// SIMATIC S7-200 SMART project (STEP 7-Micro/WIN SMART), CPU SR40

SYMBOL_TABLE 系统符号
Always_On        SM0.0    // 始终接通
Clock_1s         SM0.5    // 针对 1 s 的周期时间，时钟脉冲接通 0.5 s，断开 0.5 s.
END_SYMBOL_TABLE

ORGANIZATION_BLOCK MAIN:OB1
TITLE=程序注释
BEGIN
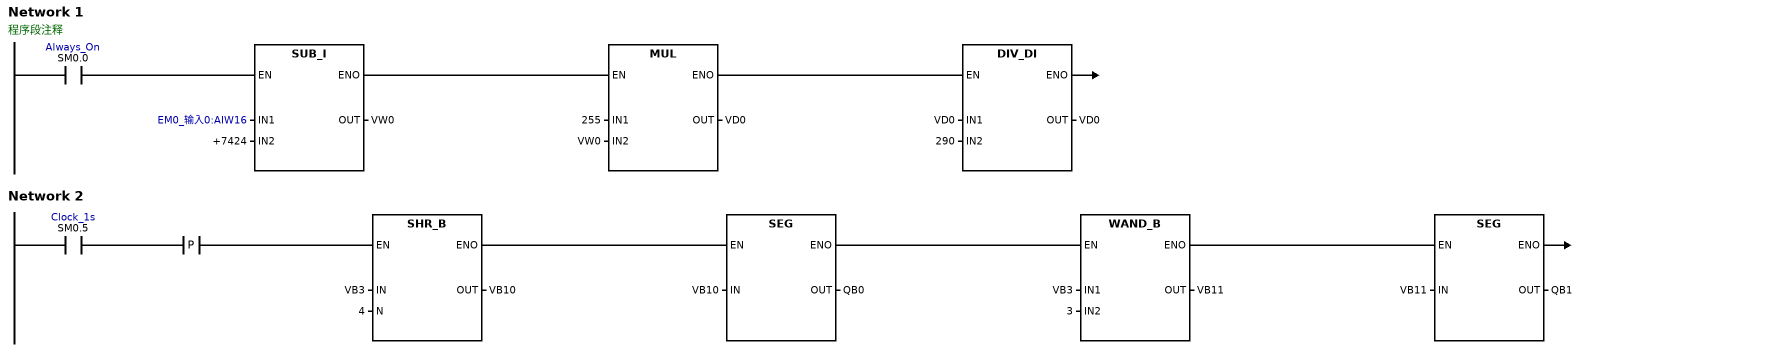
Network 1
// 程序段注释
LD     Always_On:SM0.0
MOVW   EM0_输入0:AIW16, VW0
AENO
-I     +7424, VW0
AENO
MOVW   255, VW2
AENO
MUL    VW0, VD0
AENO
/D     290, VD0
Network 2
LD     Clock_1s:SM0.5
EU
MOVB   VB3, VB10
AENO
SRB    VB10, 4
AENO
SEG    VB10, QB0
AENO
MOVB   VB3, VB11
AENO
ANDB   3, VB11
AENO
SEG    VB11, QB1
END_ORGANIZATION_BLOCK
